{attribute 'linkalways'} 
{attribute 'no_explicit_call' := 'This FB is a CLASS and must be accessed using methods or properties'}
{attribute 'enable_dynamic_creation'}
FUNCTION_BLOCK Node_F_VN_MaxElementElementwise_LREAL EXTENDS VisionNode
VAR
    ipContainer : _ITcVnContainer;
    fMax : _LREAL(0.0);
    hrPrev : _HRESULT(S_OK);
    hresult : _HRESULT(S_OK);
END_VAR

METHOD PUBLIC  Clone : I_Node
VAR
	pNode : POINTER TO Node_F_VN_MaxElementElementwise_LREAL;
END_VAR
pNode := __NEW(Node_F_VN_MaxElementElementwise_LREAL);
Clone := pNode^;
END_METHOD

METHOD FB_init : BOOL
VAR_INPUT
	bInitRetains : BOOL; // if TRUE, the retain variables are initialized (warm start / cold start)
	bInCopyCode : BOOL;  // if TRUE, the instance afterwards gets moved into the copy code (online change)
END_VAR
AddInput('ipContainer', ipContainer);
AddInput('fMax', fMax);
AddInput('hrPrev', hrPrev);
AddOutput('ipContainer', ipContainer);
AddOutput('hresult',hresult);
END_METHOD

METHOD PROTECTED OnExecute : HRESULT
hresult.Value := F_VN_MaxElementElementwise_LREAL(
    ipContainer := ipContainer.Value,
    fMax := fMax.Value,
    hrPrev:= hrPrev.Value);
END_METHOD

METHOD PUBLIC PreExecutionCheck
VAR_INPUT
	Check : I_PreExecutionChecks;
END_VAR
Check.IsTrue(ipContainer.IsValid, 'ipContainer must be a valid container');
END_METHOD

END_FUNCTION_BLOCK

(* stored: Version 1.1.0.1, ProductVersion 3.1.4024.13
   POU Node_F_VN_MaxElementElementwise_LREAL: Id {2f799da3-a18e-4231-9b79-6a42b4f81366}, SpecialFunc None
   Folder Constructor: Id {2aef5db7-241a-4fe4-aa1d-09b73643d6a4}
   Method Clone: Id {2d237528-bc82-4971-94d0-a3b9cc358452}
   Method FB_init: Id {8decbaf9-18a4-4686-a544-f126d232f40d}
   Method OnExecute: Id {b6ae5cfa-e742-491f-ac90-85c6895cf693}
   Method PreExecutionCheck: Id {9c342295-0a6c-4e12-965d-ac31cea2d809} *)
